PROGRAM PRG_PowerMeasurement
VAR
	fActivePowerAbs: REAL;
	fIL1Abs: REAL;
	fIL2Abs: REAL;
	fIL3Abs: REAL;
END_VAR

fActivePowerAbs := ABS(GVL.fActivePower);
fIL1Abs := ABS(GVL.fIL1);
fIL2Abs := ABS(GVL.fIL2);
fIL3Abs := ABS(GVL.fIL3);

END_PROGRAM

(* stored: Version 1.1.0.1, ProductVersion 3.1.4024.12
   POU PRG_PowerMeasurement: Id {927e87b5-7e0a-43fe-a0fe-0f80cfa4dfec}, SpecialFunc None *)
